(* PLC project Generated.project, CODESYS CODESYS V3.5 SP19 Patch 1 *)
(* stored: creationDateTime 2026-09-14T14:47:22.367157, modificationDateTime 2026-09-14T14:47:22.367157 *)

(* ═══════════════════════════════════════════════════════════════ 🎯 ST_CycleMachineHomingHMI — Données d'échange IHM du cycle de référencement machine ─────────────────────────────────────────────────────────────── 📄 Structuration Cmd / State / Cfg , homogène avec ST_CycleHMI / ST_CycleDiveSearchHMI / ST_CycleExtractionHMI. ═══════════════════════════════════════════════════════════════ *)
TYPE ST_CycleMachineHomingHMI : STRUCT
  Cmd : ST_CycleMachineHomingCmd;
  State : ST_MachineHoming;  (* Image publiée du FB_CycleMachineHoming (SeqStep, Step, Instruction, Failed, ordres, …) *)
  Cfg : ST_CycleMachineHomingCfg;
END_STRUCT;
END_TYPE

(* ═══════════════════════════════════════════════════════════════ ⚙️ ST_CycleMachineHomingCfg — Réglages IHM du cycle de référencement machine ─────────────────────────────────────────────────────────────── 🎯 Mise en service. Les réglages géométriques (positions capteur, offsets benne) restent portés par GVL_PERSISTENT (_WinchM1CfgPersist / _BucketCfgPersist). 💾 Ponté vers persist (_CycleMachineHomingCfgPersist) via FB_CfgPersistBridge_CycleMachineHomingCfg. ═══════════════════════════════════════════════════════════════ *)
TYPE ST_CycleMachineHomingCfg : STRUCT
  ForceStepTarget : INT := 0;  (* 🔧 Step GRAFCET cible du forçage (0=HX0 .. 9=HXF), borné côté FB *)
  Initialized : BOOL := FALSE;  (* 🚦 flag restauration boot *)
END_STRUCT;
END_TYPE

(* ═══════════════════════════════════════════════════════════════ 🎮 ST_CycleMachineHomingCmd — Commandes IHM du cycle de référencement machine ─────────────────────────────────────────────────────────────── 🎯 Cycle homing machine (FB_CycleMachineHoming) — orchestré en MAINT_N2. Séparé de ST_CycleCmd (cycle SEMI_AUTO) et de ST_ModesCmd (modes de marche). Boutons momentanés uniquement ; réglages -> ST_CycleMachineHomingCfg. ═══════════════════════════════════════════════════════════════ *)
TYPE ST_CycleMachineHomingCmd : STRUCT
  BtnStart : BOOL;  (* ▶️ Lancer le cycle de homing machine (MAINT_N2, front) — alternative au motif 3 appuis joystick *)
  BtnValidate : BOOL;  (* ✅ Validation depuis IHM (front) — équivaut à 1 appui du motif 3 appuis joystick *)
  BtnAbort : BOOL;  (* ⏹️ Quitter / abandonner le cycle homing (front) — retour HX0 sans mouvement *)
  TglCommissioning : BOOL := FALSE;  (* 🔧 Case mise en service : déverrouille le forçage de step (MAINT_N2). NON persisté (reset au reboot = sûr). *)
  BtnForceStepApply : BOOL;  (* 🔧 Applique le forçage de step (front) — impulsion ; cible = ST_CycleMachineHomingCfg.ForceStepTarget *)
END_STRUCT;
END_TYPE

(* ======================================================================= 🧭 ST_MachineHoming — Etat publie du homing conjoint machine (M1/M2/benne) ─────────────────────────────────────────────────────────────── 🎯 Rôle : Regroupe les 8 sorties homing a plat de PRG_02_Acquisition en un bus struct unique, publie sur le bus inter-PRG. 🔒 Sécurité : Homed = qualification conjointe reference machine (gate SEMI_AUTO). HomingLoss = perte reference en mouvement : arret controle SafeStop. 📄 Doc métier : DOC/AF/AF_Partie-09_Fonction_Encoder_v2.4.md (F09.08) ======================================================================= *)
TYPE ST_MachineHoming : STRUCT
  Homed : BOOL;  (* Qualification conjointe reference machine *)
  SetPosBucketOpen : BOOL;  (* Valider position actuelle = reference benne ouverte *)
  SetPosBucketClose : BOOL;  (* Valider position actuelle = reference benne fermee *)
  Active : BOOL;  (* Homing conjoint en cours *)
  HomingLoss : BOOL;  (* Perte reference en mouvement : arret controle SafeStop *)
  Step : INT;  (* Etape guidee reference (echelle de priorite E_MachineHomingStep) *)
  Instruction : STRING(120);  (* Consigne IHM reference *)
  Failed : BOOL;  (* Transaction reference abandonnee *)
  SeqStep : INT;  (* Step GRAFCET courant (E_MachineHomingTxState HX0..HXF) *)
  M3Locked : BOOL;  (* Translation M3 interdite pendant le cycle de homing machine *)
  CmdWinchM1 : ST_ProgramWinchRequest;  (* Ordre treuil M1 couple palier 1 (HX2 montee / HX3 descente) *)
  CmdWinchM2 : ST_ProgramWinchRequest;  (* Ordre treuil M2 couple palier 1 (HX2 montee / HX3 descente) *)
  CmdBucketOpen : BOOL;  (* Ordre ouverture benne palier 1 sans FDC soft *)
  CmdBucketClose : BOOL;  (* Ordre fermeture benne palier 1 sans FDC soft (HX1) *)
  CmdWinchSelect : INT;  (* Override selecteur treuil cycle homing (-1=neutre, 0=couple, 2=benne) *)
  AllowAscent : BOOL;  (* Autorisation montee par etape GRAFCET homing *)
  AllowDescend : BOOL;  (* Autorisation descente par etape GRAFCET homing *)
  SoftLimitsOff : BOOL;  (* Inhibition limites soft position (HX1..HX3 uniquement, hors capteur TOP) *)
  BucketRefInvalidate : BOOL;  (* Revoque reference benne sur abandon cycle avant HX4 *)
  ProvisionalActive : BOOL;  (* TRUE tant que le zero 0m HX1 est provisoire avant HX4 8.5m *)
  TopContactLatched : BOOL;  (* Contact TOP touche pendant cycle homing : degagement requis *)
  TopContactCount : UINT;  (* Nombre de contacts capteur TOP pendant cycle homing (purge Reset) *)
  ActionText : STRING(120);  (* Consigne d action directe du GRAFCET pour bandeau operateur *)
END_STRUCT;
END_TYPE

(* ======================================================================= 🔌 ST_ProgramWinchRequest — Demande de mouvement treuil par le programme ─────────────────────────────────────────────────────────────── 🎯 Rôle : Regroupe les demandes logiques de treuil formulées par le séquenceur 📄 Référentiel : DOC/WFLOW/CONTRACTS/INTERPRG_CONTRACT_PRG03_MODES_CYCLE_v1.0.md ======================================================================= *)
TYPE ST_ProgramWinchRequest : STRUCT
  RunRequest : BOOL;  (* Ordre marche demandé par le programme *)
  ReqAscent : BOOL;  (* Demande montée *)
  ReqDescend : BOOL;  (* Demande descente *)
  StepTgt : INT;  (* Palier de vitesse cible demandé (1 à 5, 0 = arrêt) *)
END_STRUCT;
END_TYPE
